FUNCTION_BLOCK System_NoOutput (* Composite Function Block Type *)
  (* Standard: 61499-2 *)
  (* Version 0.0, 9/19/2014, Администратор, nxtControl GmbH, template *)
  PACKAGE Main;
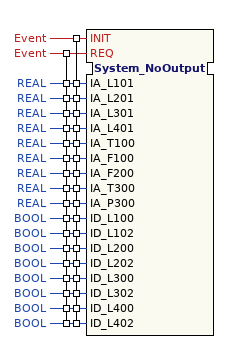
  EVENT_INPUT
    INIT WITH IA_L101, IA_L201, IA_L301, IA_L401, IA_T100, IA_F100, IA_F200, IA_T300, IA_P300, ID_L100, ID_L102, ID_L200, ID_L202, ID_L300, ID_L302, ID_L400, ID_L402;
    REQ WITH IA_L101, IA_L201, IA_L301, IA_L401, IA_T100, IA_F100, IA_F200, IA_T300, IA_P300, ID_L100, ID_L102, ID_L200, ID_L202, ID_L300, ID_L302, ID_L400, ID_L402;
  END_EVENT
  VAR_INPUT
    IA_L101 : REAL;
    IA_L201 : REAL;
    IA_L301 : REAL;
    IA_L401 : REAL;
    IA_T100 : REAL;
    IA_F100 : REAL;
    IA_F200 : REAL;
    IA_T300 : REAL;
    IA_P300 : REAL;
    ID_L100 : BOOL;
    ID_L102 : BOOL;
    ID_L200 : BOOL;
    ID_L202 : BOOL;
    ID_L300 : BOOL;
    ID_L302 : BOOL;
    ID_L400 : BOOL;
    ID_L402 : BOOL;
  END_VAR
  FBS
    T100WaterLevel : Service_ADIMeasure(PRESET_HH := 270.0, PRESET_H := 240.0, PRESET_L := 180.0, PRESET_LL := 160.0, PRESET_MINAI := 848.0, PRESET_MAXAI := 17844.0);
    T200WaterLevel : Service_ADIMeasure(PRESET_HH := 285.0, PRESET_H := 255.0, PRESET_L := 70.0, PRESET_LL := 40.0, PRESET_MINAI := 0, PRESET_MAXAI := 300.0);
    T300WaterLevel : Service_ADIMeasure(PRESET_HH := 285.0, PRESET_H := 255.0, PRESET_L := 70.0, PRESET_LL := 40.0, PRESET_MINAI := 0.0, PRESET_MAXAI := 300.0);
    T400WaterLevel : Service_ADIMeasure(PRESET_HH := 285.0, PRESET_H := 255.0, PRESET_L := 70.0, PRESET_LL := 40.0, PRESET_MINAI := 892.0, PRESET_MAXAI := 17723.0);
    T100Temperature : Service_AIMeasure(PRESET_HH := 45.0, PRESET_H := 40.0, PRESET_L := 25.0, PRESET_LL := 20.0, PRESET_MINAI := 0.0, PRESET_MAXAI := 100.0);
    F100Flow : Service_AIMeasure(PRESET_HH := 2.0, PRESET_H := 1.95, PRESET_L := 0.1, PRESET_LL := 0.0, PRESET_MINAI := 0.0, PRESET_MAXAI := 2.5);
    F200Flow : Service_AIMeasure(PRESET_HH := 2.0, PRESET_H := 1.95, PRESET_L := 0.1, PRESET_LL := 0.0, PRESET_MINAI := 0.0, PRESET_MAXAI := 2.5);
    T300Temperature : Service_AIMeasure(PRESET_HH := 45.0, PRESET_H := 40.0, PRESET_L := 25.0, PRESET_LL := 20.0, PRESET_MINAI := 0.0, PRESET_MAXAI := 100.0);
    P300Pressure : Service_AIMeasure(PRESET_HH := 0.25, PRESET_H := 0.2, PRESET_L := 0.1, PRESET_LL := 0.0, PRESET_MINAI := 0, PRESET_MAXAI := 0.25);
    T100TankControl : FB_TankControl(TempSensorIsConfigured := TRUE, PressureSensorIsConfigured := FALSE, PressureSensorHHAlarm := FALSE, PressureSensorHealthy := FALSE, WaterLevelSensorHighIsConfigured := TRUE, WaterLevelSensorLowIsConfigured := TRUE, WaterLevelSensorOverflowIsConfigured := FALSE, WaterLevelSensorOverflowAlarm := FALSE, WaterLevelSensorOverflowHealthy := FALSE);
    T200TankControl : FB_TankControl(WaterLevelSensorHighIsConfigured := TRUE, WaterLevelSensorLowIsConfigured := TRUE, TempSensorIsConfigured := FALSE, TempSensorHHAlarm := FALSE, TempSensorHealthy := FALSE, PressureSensorIsConfigured := FALSE, PressureSensorHHAlarm := FALSE, PressureSensorHealthy := FALSE, WaterLevelSensorOverflowIsConfigured := FALSE, WaterLevelSensorOverflowAlarm := FALSE, WaterLevelSensorOverflowHealthy := FALSE);
    T300TankControl : FB_TankControl(TempSensorIsConfigured := TRUE, PressureSensorIsConfigured := TRUE, WaterLevelSensorHighIsConfigured := TRUE, WaterLevelSensorLowIsConfigured := TRUE, WaterLevelSensorOverflowIsConfigured := FALSE, WaterLevelSensorOverflowAlarm := FALSE, WaterLevelSensorOverflowHealthy := FALSE);
    T400TankControl : FB_TankControl(WaterLevelSensorLowIsConfigured := TRUE, PressureSensorHealthy := FALSE, TempSensorIsConfigured := FALSE, TempSensorHHAlarm := FALSE, TempSensorHealthy := FALSE, PressureSensorIsConfigured := FALSE, PressureSensorHHAlarm := FALSE, WaterLevelSensorHighIsConfigured := TRUE, WaterLevelSensorOverflowIsConfigured := FALSE, WaterLevelSensorOverflowAlarm := FALSE, WaterLevelSensorOverflowHealthy := FALSE);
    M100PumpPIDControl : FB_PIDControl(AutoMode := TRUE, SP := 2.0, gain := 1.0, rate := 1.0, reset := 1.0, sample := 1.5);
    M200PumpPIDControl : FB_PIDControl(AutoMode := TRUE, SP := 2.0, gain := 1.0, rate := 1.0, reset := 1.0, sample := 1.5);
    WaterProcessSequenceControl : FB_SequenceControl(FillingSeqEnable := FALSE, StartSeqEnable := FALSE, ShutdownSeqEnable := FALSE, EmptyingSeqEnable := FALSE);
    WaterProcessInterlockControl : FB_InterlockControl;
    E100HeaterControl : FB_HeaterControl;
    M100PumpControl : FB_PumpControl(RangeOutMin := 0.0, RangeOutMax := 100.0);
    M200PumpControl : FB_PumpControl(RangeOutMin := 0.0, RangeOutMax := 100.0);
    Y101ValveControl : FB_ValveControl(IsControlValve := FALSE, RangeOutMin := 0.0, RangeOutMax := 0.0, RequestValue := 0.0);
    Y102ValveControl : FB_ValveControl(RangeOutMin := 0.0, IsControlValve := TRUE, RangeOutMax := 25630.0);
    Y103ValveControl : FB_ValveControl(IsControlValve := FALSE, RangeOutMin := 0.0, RangeOutMax := 0.0, RequestValue := 0.0);
    Y105ValveControl : FB_ValveControl(IsControlValve := FALSE, RangeOutMin := 0.0, RangeOutMax := 0.0, RequestValue := 0.0);
    Y201ValveControl : FB_ValveControl(IsControlValve := TRUE, RangeOutMin := 0.0, RangeOutMax := 25630.0);
    Y202ValveControl : FB_ValveControl(IsControlValve := FALSE, RangeOutMin := 0.0, RangeOutMax := 0.0, RequestValue := 0.0);
    Y203ValveControl : FB_ValveControl(IsControlValve := FALSE, RangeOutMin := 0.0, RangeOutMax := 0.0, RequestValue := 0.0);
    Y204ValveControl : FB_ValveControl(IsControlValve := FALSE, RangeOutMin := 0.0, RangeOutMax := 0.0, RequestValue := 0.0);
    Y501ValveControl : FB_ValveControl(IsControlValve := FALSE, RangeOutMin := 0.0, RangeOutMax := 0.0, RequestValue := 0.0);
    Y404ValveControl : FB_ValveControl(IsControlValve := FALSE, RangeOutMin := 0.0, RangeOutMax := 0.0, RequestValue := 0.0);
    Y401ValveControl : FB_ValveControl(IsControlValve := FALSE, RangeOutMin := 0.0, RangeOutMax := 0.0, RequestValue := 0.0);
    Y303ValveControl : FB_ValveControl(IsControlValve := FALSE, RangeOutMin := 0.0, RangeOutMax := 0.0, RequestValue := 0.0);
    Y403ValveControl : FB_ValveControl(IsControlValve := FALSE, RangeOutMin := 0.0, RangeOutMax := 0.0, RequestValue := 0.0);
    Y402ValveControl : FB_ValveControl(IsControlValve := FALSE, RangeOutMin := 0.0, RangeOutMax := 0.0, RequestValue := 0.0);
    Y305ValveControl : FB_ValveControl(IsControlValve := FALSE, RangeOutMin := 0.0, RangeOutMax := 0.0, RequestValue := 0.0);
    Y302ValveControl : FB_ValveControl(IsControlValve := FALSE, RangeOutMin := 0.0, RangeOutMax := 0.0, RequestValue := 0.0);
    Y301ValveControl : FB_ValveControl(IsControlValve := FALSE, RangeOutMin := 0.0, RangeOutMax := 0.0, RequestValue := 0.0);
    M100Control : Service_AOControl(OM := FALSE, OM_Value := 0.0);
    M200Control : Service_AOControl(OM := FALSE, OM_Value := 0.0);
    Y102Control : Service_AOControl(OM := FALSE, OM_Value := 0.0);
    Y201Control : Service_AOControl(OM := FALSE, OM_Value := 0.0);
    E100Control : Service_DOControl(OM := FALSE, OM_ON := FALSE);
    Y101Control : Service_DOControl(OM := FALSE, OM_ON := FALSE);
    Y103Control : Service_DOControl(OM := FALSE, OM_ON := FALSE);
    Y105Control : Service_DOControl(OM := FALSE, OM_ON := FALSE);
    Y202Control : Service_DOControl(OM := FALSE, OM_ON := FALSE);
    Y203Control : Service_DOControl(OM := FALSE, OM_ON := FALSE);
    Y204Control : Service_DOControl(OM := FALSE, OM_ON := FALSE);
    Y301Control : Service_DOControl(OM := FALSE, OM_ON := FALSE);
    Y302Control : Service_DOControl(OM := FALSE, OM_ON := FALSE);
    Y303Control : Service_DOControl(OM := FALSE, OM_ON := FALSE);
    Y305Control : Service_DOControl(OM := FALSE, OM_ON := FALSE);
    Y401Control : Service_DOControl(OM := FALSE, OM_ON := FALSE);
    Y402Control : Service_DOControl(OM := FALSE, OM_ON := FALSE);
    Y403Control : Service_DOControl(OM := FALSE, OM_ON := FALSE);
    Y404Control : Service_DOControl(OM := FALSE, OM_ON := FALSE);
    Y501Control : Service_DOControl(OM := FALSE, OM_ON := FALSE);
    FB1 : NOT1;
    FB6 : NOT2;
    FB5 : NOT3;
    FB7 : NOT1;
    FB8 : NOT1;
    FB11 : NOT10;
    FB9 : NOT16;
  END_FBS
  EVENT_CONNECTIONS
    T100WaterLevel.INITO TO T200WaterLevel.INIT;
    T100WaterLevel.CNF TO T200WaterLevel.REQ;
    T200WaterLevel.INITO TO T300WaterLevel.INIT;
    T300WaterLevel.INITO TO T400WaterLevel.INIT;
    T200WaterLevel.CNF TO T300WaterLevel.REQ;
    T300WaterLevel.CNF TO T400WaterLevel.REQ;
    T400WaterLevel.INITO TO T100Temperature.INIT;
    T400WaterLevel.CNF TO T100Temperature.REQ;
    T100Temperature.INITO TO F100Flow.INIT;
    T100Temperature.CNF TO F100Flow.REQ;
    F100Flow.INITO TO F200Flow.INIT;
    F100Flow.CNF TO F200Flow.REQ;
    F200Flow.INITO TO T300Temperature.INIT;
    F200Flow.CNF TO T300Temperature.REQ;
    T300Temperature.INITO TO P300Pressure.INIT;
    T300Temperature.CNF TO P300Pressure.REQ;
    P300Pressure.INITO TO T100TankControl.INIT;
    P300Pressure.CNF TO FB6.REQ;
    FB6.CNF TO T100TankControl.REQ;
    T100TankControl.INITO TO T200TankControl.INIT;
    T200TankControl.INITO TO T300TankControl.INIT;
    T300TankControl.INITO TO T400TankControl.INIT;
    T100TankControl.CNF TO FB1.REQ;
    T200TankControl.CNF TO FB5.REQ;
    FB5.CNF TO T300TankControl.REQ;
    T300TankControl.CNF TO FB7.REQ;
    FB7.CNF TO T400TankControl.REQ;
    T400TankControl.INITO TO M100PumpPIDControl.INIT;
    T400TankControl.CNF TO M100PumpPIDControl.REQ;
    M100PumpPIDControl.INITO TO M200PumpPIDControl.INIT;
    M100PumpPIDControl.CNF TO M200PumpPIDControl.REQ;
    M200PumpPIDControl.INITO TO WaterProcessSequenceControl.INIT;
    WaterProcessSequenceControl.INITO TO WaterProcessInterlockControl.INIT;
    WaterProcessInterlockControl.INITO TO E100HeaterControl.INIT;
    WaterProcessInterlockControl.CNF TO E100HeaterControl.REQ;
    E100HeaterControl.INITO TO M100PumpControl.INIT;
    E100HeaterControl.CNF TO M100PumpControl.REQ;
    M100PumpControl.INITO TO M200PumpControl.INIT;
    M100PumpControl.CNF TO M200PumpControl.REQ;
    M200PumpControl.INITO TO Y101ValveControl.INIT;
    M200PumpControl.CNF TO Y101ValveControl.REQ;
    Y101ValveControl.INITO TO Y102ValveControl.INIT;
    Y101ValveControl.CNF TO Y102ValveControl.REQ;
    Y102ValveControl.INITO TO Y103ValveControl.INIT;
    Y102ValveControl.CNF TO Y103ValveControl.REQ;
    Y103ValveControl.INITO TO Y105ValveControl.INIT;
    Y103ValveControl.CNF TO Y105ValveControl.REQ;
    Y105ValveControl.INITO TO Y201ValveControl.INIT;
    Y105ValveControl.CNF TO Y201ValveControl.REQ;
    Y201ValveControl.INITO TO Y202ValveControl.INIT;
    Y201ValveControl.CNF TO Y202ValveControl.REQ;
    Y202ValveControl.INITO TO Y203ValveControl.INIT;
    Y202ValveControl.CNF TO Y203ValveControl.REQ;
    Y203ValveControl.INITO TO Y204ValveControl.INIT;
    Y203ValveControl.CNF TO Y204ValveControl.REQ;
    Y204ValveControl.INITO TO Y301ValveControl.INIT;
    Y204ValveControl.CNF TO Y301ValveControl.REQ;
    Y301ValveControl.INITO TO Y302ValveControl.INIT;
    Y301ValveControl.CNF TO Y302ValveControl.REQ;
    Y302ValveControl.INITO TO Y303ValveControl.INIT;
    Y302ValveControl.CNF TO Y303ValveControl.REQ;
    Y303ValveControl.INITO TO Y305ValveControl.INIT;
    Y303ValveControl.CNF TO Y305ValveControl.REQ;
    Y305ValveControl.INITO TO Y401ValveControl.INIT;
    Y305ValveControl.CNF TO Y401ValveControl.REQ;
    Y401ValveControl.INITO TO Y402ValveControl.INIT;
    Y401ValveControl.CNF TO Y402ValveControl.REQ;
    Y402ValveControl.INITO TO Y403ValveControl.INIT;
    Y402ValveControl.CNF TO Y403ValveControl.REQ;
    Y403ValveControl.INITO TO Y404ValveControl.INIT;
    Y403ValveControl.CNF TO Y404ValveControl.REQ;
    Y404ValveControl.INITO TO Y501ValveControl.INIT;
    Y404ValveControl.CNF TO Y501ValveControl.REQ;
    M200PumpPIDControl.CNF TO FB11.REQ;
    FB11.CNF TO WaterProcessSequenceControl.REQ;
    WaterProcessSequenceControl.CNF TO FB9.REQ;
    FB9.CNF TO FB8.REQ;
    FB8.CNF TO WaterProcessInterlockControl.REQ;
    Y501ValveControl.INITO TO M100Control.INIT;
    Y501ValveControl.CNF TO M100Control.REQ;
    M100Control.INITO TO M200Control.INIT;
    M100Control.CNF TO M200Control.REQ;
    M200Control.INITO TO Y102Control.INIT;
    M200Control.CNF TO Y102Control.REQ;
    Y102Control.INITO TO Y201Control.INIT;
    Y102Control.CNF TO Y201Control.REQ;
    Y201Control.INITO TO E100Control.INIT;
    Y201Control.CNF TO E100Control.REQ;
    Y204Control.INITO TO Y301Control.INIT;
    Y204Control.CNF TO Y301Control.REQ;
    E100Control.INITO TO Y101Control.INIT;
    E100Control.CNF TO Y101Control.REQ;
    Y101Control.INITO TO Y103Control.INIT;
    Y101Control.CNF TO Y103Control.REQ;
    Y103Control.INITO TO Y105Control.INIT;
    Y103Control.CNF TO Y105Control.REQ;
    Y105Control.INITO TO Y202Control.INIT;
    Y105Control.CNF TO Y202Control.REQ;
    Y202Control.INITO TO Y203Control.INIT;
    Y202Control.CNF TO Y203Control.REQ;
    Y203Control.INITO TO Y204Control.INIT;
    Y203Control.CNF TO Y204Control.REQ;
    Y301Control.INITO TO Y302Control.INIT;
    Y301Control.CNF TO Y302Control.REQ;
    Y302Control.INITO TO Y303Control.INIT;
    Y302Control.CNF TO Y303Control.REQ;
    Y303Control.INITO TO Y305Control.INIT;
    Y303Control.CNF TO Y305Control.REQ;
    Y305Control.INITO TO Y401Control.INIT;
    Y305Control.CNF TO Y401Control.REQ;
    Y401Control.INITO TO Y402Control.INIT;
    Y401Control.CNF TO Y402Control.REQ;
    Y402Control.INITO TO Y403Control.INIT;
    Y402Control.CNF TO Y403Control.REQ;
    Y403Control.INITO TO Y404Control.INIT;
    Y403Control.CNF TO Y404Control.REQ;
    Y404Control.INITO TO Y501Control.INIT;
    Y404Control.CNF TO Y501Control.REQ;
    INIT TO T100WaterLevel.INIT;
    FB1.CNF TO T200TankControl.REQ;
    REQ TO T100WaterLevel.REQ;
  END_CONNECTIONS
  DATA_CONNECTIONS
    ID_L100 TO T100WaterLevel.DIH;
    ID_L102 TO T100WaterLevel.DIL;
    ID_L200 TO T200WaterLevel.DIH;
    ID_L202 TO T200WaterLevel.DIL;
    ID_L300 TO T300WaterLevel.DIH;
    ID_L302 TO T300WaterLevel.DIL;
    ID_L400 TO T400WaterLevel.DIH;
    ID_L402 TO T400WaterLevel.DIL;
    IA_F100 TO F100Flow.AI;
    IA_F200 TO F200Flow.AI;
    T100WaterLevel.SensorFault TO FB6.IN1;
    T100Temperature.SensorFault TO FB6.IN2;
    FB6.OUT1 TO T100TankControl.WaterLevelSensorHighHealthy;
    FB6.OUT2 TO T100TankControl.TempSensorHealthy;
    T100WaterLevel.AlarmLL TO T100TankControl.WaterLevelSensorLLAlarm;
    FB6.OUT1 TO T100TankControl.WaterLevelSensorLowHealthy;
    T200WaterLevel.SensorFault TO FB1.IN1;
    FB1.OUT1 TO T200TankControl.WaterLevelSensorHighHealthy;
    FB1.OUT1 TO T200TankControl.WaterLevelSensorLowHealthy;
    T200WaterLevel.AlarmHH TO T200TankControl.WaterLevelSensorHHAlarm;
    T200WaterLevel.AlarmLL TO T200TankControl.WaterLevelSensorLLAlarm;
    T300WaterLevel.SensorFault TO FB5.IN1;
    FB5.OUT1 TO T300TankControl.WaterLevelSensorHighHealthy;
    FB5.OUT1 TO T300TankControl.WaterLevelSensorLowHealthy;
    T300Temperature.SensorFault TO FB5.IN2;
    FB5.OUT2 TO T300TankControl.TempSensorHealthy;
    P300Pressure.SensorFault TO FB5.IN3;
    FB5.OUT3 TO T300TankControl.PressureSensorHealthy;
    T300Temperature.AlarmHH TO T300TankControl.TempSensorHHAlarm;
    P300Pressure.AlarmHH TO T300TankControl.PressureSensorHHAlarm;
    T300WaterLevel.AlarmHH TO T300TankControl.WaterLevelSensorHHAlarm;
    T300WaterLevel.AlarmLL TO T300TankControl.WaterLevelSensorLLAlarm;
    T400WaterLevel.SensorFault TO FB7.IN1;
    FB7.OUT1 TO T400TankControl.WaterLevelSensorHighHealthy;
    FB7.OUT1 TO T400TankControl.WaterLevelSensorLowHealthy;
    T100WaterLevel.AlarmHH TO T100TankControl.WaterLevelSensorHHAlarm;
    T100Temperature.AlarmHH TO T100TankControl.TempSensorHHAlarm;
    T400WaterLevel.AlarmHH TO T400TankControl.WaterLevelSensorHHAlarm;
    T400WaterLevel.AlarmLL TO T400TankControl.WaterLevelSensorLLAlarm;
    IA_F100 TO M100PumpPIDControl.PV;
    IA_F200 TO M200PumpPIDControl.PV;
    T300TankControl.OverPresuure TO WaterProcessSequenceControl.T300_OverPressure;
    T100TankControl.InfeedEnabled TO FB11.IN1;
    T100TankControl.OutfeedEnabled TO FB11.IN2;
    T100TankControl.HeatEnabled TO FB11.IN3;
    T200TankControl.InfeedEnabled TO FB11.IN4;
    T200TankControl.OutfeedEnabled TO FB11.IN5;
    T300TankControl.InfeedEnabled TO FB11.IN6;
    T300TankControl.OutfeedEnabled TO FB11.IN7;
    T300TankControl.HeatEnabled TO FB11.IN8;
    FB11.OUT1 TO WaterProcessSequenceControl.T100_Overflow;
    FB11.OUT2 TO WaterProcessSequenceControl.T100_Underflow;
    FB11.OUT3 TO WaterProcessSequenceControl.T100_Overheat;
    FB11.OUT4 TO WaterProcessSequenceControl.T200_Overflow;
    FB11.OUT5 TO WaterProcessSequenceControl.T200_Underflow;
    FB11.OUT6 TO WaterProcessSequenceControl.T300_Overflow;
    FB11.OUT7 TO WaterProcessSequenceControl.T300_Underflow;
    FB11.OUT8 TO WaterProcessSequenceControl.T300_Overheat;
    T400TankControl.InfeedEnabled TO FB11.IN9;
    FB11.OUT9 TO WaterProcessSequenceControl.T400_Overflow;
    T400TankControl.OutfeedEnabled TO FB11.IN10;
    FB11.OUT10 TO WaterProcessSequenceControl.T400_Underflow;
    WaterProcessSequenceControl.Y101_Open TO Y101ValveControl.RequestStart;
    WaterProcessSequenceControl.Y102_Open TO Y102ValveControl.RequestStart;
    WaterProcessSequenceControl.Y103_Open TO Y103ValveControl.RequestStart;
    WaterProcessSequenceControl.Y105_Open TO Y105ValveControl.RequestStart;
    WaterProcessSequenceControl.Y201_Open TO Y201ValveControl.RequestStart;
    WaterProcessSequenceControl.Y202_Open TO Y202ValveControl.RequestStart;
    WaterProcessSequenceControl.Y203_Open TO Y203ValveControl.RequestStart;
    WaterProcessSequenceControl.Y204_Open TO Y204ValveControl.RequestStart;
    WaterProcessSequenceControl.Y301_Open TO Y301ValveControl.RequestStart;
    WaterProcessSequenceControl.Y302_Open TO Y302ValveControl.RequestStart;
    WaterProcessSequenceControl.Y303_Open TO Y303ValveControl.RequestStart;
    WaterProcessSequenceControl.Y305_Open TO Y305ValveControl.RequestStart;
    WaterProcessSequenceControl.Y401_Open TO Y401ValveControl.RequestStart;
    WaterProcessSequenceControl.Y402_Open TO Y402ValveControl.RequestStart;
    WaterProcessSequenceControl.Y403_Open TO Y403ValveControl.RequestStart;
    WaterProcessSequenceControl.Y404_Open TO Y404ValveControl.RequestStart;
    WaterProcessSequenceControl.Y501_Open TO Y501ValveControl.RequestStart;
    WaterProcessSequenceControl.E100_On TO E100HeaterControl.RequestStart;
    WaterProcessSequenceControl.M100_On TO M100PumpControl.RequestStart;
    WaterProcessSequenceControl.M200_On TO M200PumpControl.RequestStart;
    T300TankControl.OverPresuure TO WaterProcessInterlockControl.T300_OverPressure;
    T100TankControl.InfeedEnabled TO FB9.IN1;
    T100TankControl.OutfeedEnabled TO FB9.IN2;
    T100TankControl.HeatEnabled TO FB9.IN3;
    T200TankControl.InfeedEnabled TO FB9.IN4;
    T200TankControl.OutfeedEnabled TO FB9.IN5;
    T300TankControl.InfeedEnabled TO FB9.IN6;
    T300TankControl.OutfeedEnabled TO FB9.IN7;
    T300TankControl.HeatEnabled TO FB9.IN8;
    T400TankControl.InfeedEnabled TO FB9.IN9;
    T400TankControl.OutfeedEnabled TO FB9.IN10;
    Y102ValveControl.ValveOn TO FB9.IN11;
    FB9.OUT1 TO WaterProcessInterlockControl.T100_Overflow;
    FB9.OUT2 TO WaterProcessInterlockControl.T100_Underflow;
    FB9.OUT3 TO WaterProcessInterlockControl.T100_Overheat;
    FB9.OUT4 TO WaterProcessInterlockControl.T200_Overflow;
    FB9.OUT5 TO WaterProcessInterlockControl.T200_Underflow;
    FB9.OUT6 TO WaterProcessInterlockControl.T300_Overflow;
    FB9.OUT7 TO WaterProcessInterlockControl.T300_Underflow;
    FB9.OUT8 TO WaterProcessInterlockControl.T300_Overheat;
    FB9.OUT9 TO WaterProcessInterlockControl.T400_Overflow;
    FB9.OUT10 TO WaterProcessInterlockControl.T400_Underflow;
    FB9.OUT11 TO WaterProcessInterlockControl.Y102_Closed;
    Y201ValveControl.ValveOn TO FB9.IN12;
    FB9.OUT12 TO WaterProcessInterlockControl.Y201_Closed;
    Y203ValveControl.ValveOn TO FB9.IN13;
    FB9.OUT13 TO WaterProcessInterlockControl.Y203_Closed;
    Y301ValveControl.ValveOn TO FB9.IN15;
    FB9.OUT15 TO WaterProcessInterlockControl.Y301_Closed;
    Y303ValveControl.ValveOn TO FB9.IN16;
    FB9.OUT16 TO WaterProcessInterlockControl.Y303_Closed;
    FB8.OUT1 TO WaterProcessInterlockControl.Y403_Closed;
    Y403ValveControl.ValveOn TO FB8.IN1;
    WaterProcessInterlockControl.E100_On TO E100HeaterControl.ReadyToStart;
    WaterProcessInterlockControl.M100_On TO M100PumpControl.ReadyToStart;
    WaterProcessInterlockControl.M200_On TO M200PumpControl.ReadyToStart;
    M100PumpPIDControl.OUT TO M100PumpControl.RequestValue;
    M200PumpPIDControl.OUT TO M200PumpControl.RequestValue;
    WaterProcessInterlockControl.Y101_Open TO Y101ValveControl.ReadyToStart;
    WaterProcessInterlockControl.Y102_Open TO Y102ValveControl.ReadyToStart;
    WaterProcessInterlockControl.Y103_Open TO Y103ValveControl.ReadyToStart;
    WaterProcessInterlockControl.Y105_Open TO Y105ValveControl.ReadyToStart;
    WaterProcessInterlockControl.Y201_Open TO Y201ValveControl.ReadyToStart;
    WaterProcessInterlockControl.Y202_Open TO Y202ValveControl.ReadyToStart;
    WaterProcessInterlockControl.Y203_Open TO Y203ValveControl.ReadyToStart;
    WaterProcessInterlockControl.Y204_Open TO Y204ValveControl.ReadyToStart;
    WaterProcessInterlockControl.Y301_Open TO Y301ValveControl.ReadyToStart;
    WaterProcessInterlockControl.Y302_Open TO Y302ValveControl.ReadyToStart;
    WaterProcessInterlockControl.Y303_Open TO Y303ValveControl.ReadyToStart;
    WaterProcessInterlockControl.Y305_Open TO Y305ValveControl.ReadyToStart;
    WaterProcessInterlockControl.Y401_Open TO Y401ValveControl.ReadyToStart;
    WaterProcessInterlockControl.Y402_Open TO Y402ValveControl.ReadyToStart;
    WaterProcessInterlockControl.Y403_Open TO Y403ValveControl.ReadyToStart;
    WaterProcessInterlockControl.Y404_Open TO Y404ValveControl.ReadyToStart;
    WaterProcessInterlockControl.Y501_Open TO Y501ValveControl.ReadyToStart;
    M100PumpPIDControl.OUT TO Y102ValveControl.RequestValue;
    M200PumpPIDControl.OUT TO Y201ValveControl.RequestValue;
    E100HeaterControl.HeaterOn TO E100Control.CMD_ON;
    M100PumpControl.PumpValue TO M100Control.AOValue;
    M200PumpControl.PumpValue TO M200Control.AOValue;
    Y102ValveControl.ValveValue TO Y102Control.AOValue;
    Y201ValveControl.ValveValue TO Y201Control.AOValue;
    Y101ValveControl.ValveOn TO Y101Control.CMD_ON;
    Y103ValveControl.ValveOn TO Y103Control.CMD_ON;
    Y105ValveControl.ValveOn TO Y105Control.CMD_ON;
    Y202ValveControl.ValveOn TO Y202Control.CMD_ON;
    Y203ValveControl.ValveOn TO Y203Control.CMD_ON;
    Y204ValveControl.ValveOn TO Y204Control.CMD_ON;
    Y301ValveControl.ValveOn TO Y301Control.CMD_ON;
    Y302ValveControl.ValveOn TO Y302Control.CMD_ON;
    Y303ValveControl.ValveOn TO Y303Control.CMD_ON;
    Y305ValveControl.ValveOn TO Y305Control.CMD_ON;
    Y401ValveControl.ValveOn TO Y401Control.CMD_ON;
    Y402ValveControl.ValveOn TO Y402Control.CMD_ON;
    Y403ValveControl.ValveOn TO Y403Control.CMD_ON;
    Y404ValveControl.ValveOn TO Y404Control.CMD_ON;
    Y501ValveControl.ValveOn TO Y501Control.CMD_ON;
    IA_L101 TO T100WaterLevel.AI;
    IA_L201 TO T200WaterLevel.AI;
    IA_L301 TO T300WaterLevel.AI;
    IA_L401 TO T400WaterLevel.AI;
    IA_T100 TO T100Temperature.AI;
    IA_T300 TO T300Temperature.AI;
    IA_P300 TO P300Pressure.AI;
  END_CONNECTIONS
END_FUNCTION_BLOCK
